INTERFACE ITF_BaseTopElementDecoratorParent EXTENDS ITF_BaseTopElement

END_INTERFACE

(* stored: Version 1.1.0.1
   Itf ITF_BaseTopElementDecoratorParent: Id {5a77b686-f616-01f0-264a-0d7b9a187e8d} *)
